PROGRAM PRG_SignalGenerators_TEST
VAR
END_VAR

END_PROGRAM

(* stored: Version 1.1.0.1, ProductVersion 3.1.4024.13
   POU PRG_SignalGenerators_TEST: Id {069c858e-8fc4-4085-9d60-c0c54c3c4a3e}, SpecialFunc None *)
